FUNCTION_BLOCK FB_GCSpinAxisJogCWServiceTests EXTENDS TcUnit.FB_TestSuite
VAR
	Context : ST_ServiceContext;
END_VAR

Context.ModuleId := E_ModuleId.GC1;
Context.UtcDateTime := '20260813123456007';

InjectedJogErrorStopsAndReleasesAxis();
InvalidParametersAreRejectedBeforeAxisOwnership();

METHOD InjectedJogErrorStopsAndReleasesAxis
VAR_INST
	FakeAxis : FB_FakeAxis_BaseUnit;
	Axis : I_Axis_BaseUnit;
	Service : FB_GCSpinAxisJogCWServices;
	Ctrl : ST_ServiceCtrl;
	Param : ST_GCSpinAxisJogParam;
	CallRecord : ST_FakeAxisCall;
	nPhase : UINT;
END_VAR
TEST('InjectedJogErrorStopsAndReleasesAxis');

CASE nPhase OF
	0:
		FakeAxis.M_ResetScenario();
		Axis := FakeAxis;
		Param.Position := 1.5;
		Param.Velocity := 12.5;
		Param.Acceleration := 20;
		Param.Deceleration := 30;
		AssertTrue(Condition := FakeAxis.M_QueueResult(Operation := E_FakeAxisOperation.Jog, AfterActiveCycles := 2, Done := FALSE, InVelocity := FALSE, Error := TRUE, ErrorId := 16#4444), Message := 'Jog Error script must be accepted.');
		Service(Ctrl := Ctrl, Param := Param, Context := Context, Axis_BaseUnit := Axis, ResourceOwnerId := 11);
		FakeAxis.M_CyclicUpdate();
		nPhase := 1;

	1:
		Ctrl.PackMLIn.eCommand := E_PackMLCommand.Clear;
		Ctrl.PackMLIn.bCommandChangeRequest := TRUE;
		Service(Ctrl := Ctrl, Param := Param, Context := Context, Axis_BaseUnit := Axis, ResourceOwnerId := 11);
		FakeAxis.M_CyclicUpdate();
		nPhase := 2;

	2:
		Ctrl.PackMLIn.bCommandChangeRequest := FALSE;
		Service(Ctrl := Ctrl, Param := Param, Context := Context, Axis_BaseUnit := Axis, ResourceOwnerId := 11);
		FakeAxis.M_CyclicUpdate();
		Ctrl.PackMLIn.eCommand := E_PackMLCommand.Reset;
		Ctrl.PackMLIn.bCommandChangeRequest := TRUE;
		Service(Ctrl := Ctrl, Param := Param, Context := Context, Axis_BaseUnit := Axis, ResourceOwnerId := 11);
		FakeAxis.M_CyclicUpdate();
		nPhase := 3;

	3:
		Ctrl.PackMLIn.bCommandChangeRequest := FALSE;
		Service(Ctrl := Ctrl, Param := Param, Context := Context, Axis_BaseUnit := Axis, ResourceOwnerId := 11);
		FakeAxis.M_CyclicUpdate();
		Ctrl.PackMLIn.eCommand := E_PackMLCommand.Start;
		Ctrl.PackMLIn.bCommandChangeRequest := TRUE;
		Service(Ctrl := Ctrl, Param := Param, Context := Context, Axis_BaseUnit := Axis, ResourceOwnerId := 11);
		FakeAxis.M_CyclicUpdate();
		Ctrl.PackMLIn.bCommandChangeRequest := FALSE;
		AssertTrue(Condition := Service.PackMLOut.eStateCurrent = E_PackMLState.Execute, Message := 'Valid Jog must enter Execute.');
		nPhase := 4;

	4:
		Service(Ctrl := Ctrl, Param := Param, Context := Context, Axis_BaseUnit := Axis, ResourceOwnerId := 11);
		FakeAxis.M_CyclicUpdate();
		AssertTrue(Condition := FakeAxis.M_GetCall(Index := FakeAxis.HistoryCount, CallRecord => CallRecord), Message := 'Jog command must be recorded.');
		AssertTrue(Condition := CallRecord.JogForward AND NOT CallRecord.JogBackwards, Message := 'Jog direction must be forward only.');
		AssertTrue(Condition := (CallRecord.Velocity = 12.5) AND (CallRecord.Acceleration = 20) AND (CallRecord.Deceleration = 30), Message := 'Jog parameters must reach the Axis unchanged.');
		nPhase := 5;

	5:
		Service(Ctrl := Ctrl, Param := Param, Context := Context, Axis_BaseUnit := Axis, ResourceOwnerId := 11);
		FakeAxis.M_CyclicUpdate();
		AssertTrue(Condition := Service.Status.ErrorList[1].MainErrorId = 0, Message := 'Jog Error must still be pending after one active cycle.');
		nPhase := 6;

	6:
		Service(Ctrl := Ctrl, Param := Param, Context := Context, Axis_BaseUnit := Axis, ResourceOwnerId := 11);
		FakeAxis.M_CyclicUpdate();
		AssertTrue(Condition := Service.Status.ErrorList[1].MainErrorId = E_GCServiceErrorCode.Axis_Command_Error_During_Execute, Message := 'Jog Error must use the shared Service error code.');
		AssertTrue(Condition := Service.Status.ErrorList[1].SourceErrorId = 16#4444, Message := 'Jog Error must preserve the Axis source error ID.');
		AssertTrue(Condition := Service.Status.ErrorList[1].ModuleId = Context.ModuleId, Message := 'Jog Error must preserve the injected Module ID.');
		AssertTrue(Condition := Service.Status.ErrorList[1].DateTime = Context.UtcDateTime, Message := 'Jog Error must preserve the injected UTC timestamp.');
		AssertTrue(Condition := Service.Status.ErrorList[1].Severity = E_Severity.Alarm, Message := 'Jog Error must use Alarm severity.');
		AssertTrue(Condition := Service.Status.ServiceErrorId = 0, Message := 'Jog must not update ServiceErrorId.');
		nPhase := 7;

	7:
		Service(Ctrl := Ctrl, Param := Param, Context := Context, Axis_BaseUnit := Axis, ResourceOwnerId := 11);
		FakeAxis.M_CyclicUpdate();
		AssertTrue(Condition := Service.PackMLOut.eStateCurrent = E_PackMLState.Stopped, Message := 'Jog Error must finish the Stop transition.');
		AssertFalse(Condition := Axis.M_IsResourceOwner(OwnerId := 11), Message := 'Jog Stop must release ownership.');
		AssertTrue(Condition := FakeAxis.M_GetCall(Index := FakeAxis.HistoryCount, CallRecord => CallRecord), Message := 'Jog cancellation must be recorded.');
		AssertFalse(Condition := CallRecord.JogForward OR CallRecord.JogBackwards, Message := 'Stopping must cancel both Jog directions.');
		nPhase := 0;
		TEST_FINISHED();
END_CASE
END_METHOD

METHOD InvalidParametersAreRejectedBeforeAxisOwnership
VAR_INST
	FakeAxis : FB_FakeAxis_BaseUnit;
	Axis : I_Axis_BaseUnit;
	Service : FB_GCSpinAxisJogCWServices;
	Ctrl : ST_ServiceCtrl;
	Param : ST_GCSpinAxisJogParam;
	nPhase : UINT;
END_VAR
TEST('InvalidParametersAreRejectedBeforeAxisOwnership');

CASE nPhase OF
	0:
		FakeAxis.M_ResetScenario();
		Axis := FakeAxis;
		Param.Velocity := 0;
		Service(Ctrl := Ctrl, Param := Param, Context := Context, Axis_BaseUnit := Axis, ResourceOwnerId := 12);
		FakeAxis.M_CyclicUpdate();
		nPhase := 1;
	1:
		Ctrl.PackMLIn.eCommand := E_PackMLCommand.Clear;
		Ctrl.PackMLIn.bCommandChangeRequest := TRUE;
		Service(Ctrl := Ctrl, Param := Param, Context := Context, Axis_BaseUnit := Axis, ResourceOwnerId := 12);
		FakeAxis.M_CyclicUpdate();
		Ctrl.PackMLIn.bCommandChangeRequest := FALSE;
		Service(Ctrl := Ctrl, Param := Param, Context := Context, Axis_BaseUnit := Axis, ResourceOwnerId := 12);
		FakeAxis.M_CyclicUpdate();
		Ctrl.PackMLIn.eCommand := E_PackMLCommand.Reset;
		Ctrl.PackMLIn.bCommandChangeRequest := TRUE;
		Service(Ctrl := Ctrl, Param := Param, Context := Context, Axis_BaseUnit := Axis, ResourceOwnerId := 12);
		FakeAxis.M_CyclicUpdate();
		nPhase := 2;
	2:
		Ctrl.PackMLIn.bCommandChangeRequest := FALSE;
		Service(Ctrl := Ctrl, Param := Param, Context := Context, Axis_BaseUnit := Axis, ResourceOwnerId := 12);
		FakeAxis.M_CyclicUpdate();
		Ctrl.PackMLIn.eCommand := E_PackMLCommand.Start;
		Ctrl.PackMLIn.bCommandChangeRequest := TRUE;
		Service(Ctrl := Ctrl, Param := Param, Context := Context, Axis_BaseUnit := Axis, ResourceOwnerId := 12);
		FakeAxis.M_CyclicUpdate();
		AssertTrue(Condition := Service.Status.ErrorList[1].MainErrorId = E_GCServiceErrorCode.Invalid_Param, Message := 'Zero Jog velocity must be rejected as Invalid_Param.');
		AssertTrue(Condition := Service.Status.ErrorList[1].SourceErrorId = 0, Message := 'Invalid Jog data must use source ID zero.');
		AssertTrue(Condition := Service.Status.ErrorList[1].ModuleId = Context.ModuleId, Message := 'Invalid Jog data must preserve the injected Module ID.');
		AssertTrue(Condition := Service.Status.ErrorList[1].DateTime = Context.UtcDateTime, Message := 'Invalid Jog data must preserve the injected UTC timestamp.');
		AssertTrue(Condition := Service.Status.ServiceErrorId = 0, Message := 'Invalid Jog data must not update ServiceErrorId.');
		AssertFalse(Condition := Axis.M_IsResourceOwner(OwnerId := 12), Message := 'Parameter validation must occur before ownership.');
		nPhase := 0;
		TEST_FINISHED();
END_CASE
END_METHOD

END_FUNCTION_BLOCK

(* stored: Version 1.1.0.1, ProductVersion 3.1.4026.18
   POU FB_GCSpinAxisJogCWServiceTests: Id {66d53592-ab9f-4c39-a5ad-9cf4021704bb}, SpecialFunc None
   Method InjectedJogErrorStopsAndReleasesAxis: Id {a66861a0-b183-421d-8878-c312f33c87bf}
   Method InvalidParametersAreRejectedBeforeAxisOwnership: Id {bedc1917-f303-4b09-9d7b-ad3776ea7d15} *)
